{attribute 'GeneratedUsingTerminal: EL6201-0000-0017'}
{attribute addProperty BoxType "EL6201-0000-0017"}
{attribute addProperty Id "Slave_29A_DI0BOOL1Slave_29A_DI1BOOL1Slave_29A_DI2BOOL1Slave_29A_DI3BOOL1Slave_29B_DI0BOOL1Slave_29B_DI1BOOL1Slave_29B_DI2BOOL1Slave_29B_DI3BOOL1"}
{attribute addProperty CRC "3259051410"}
{attribute addProperty Size "8"}
TYPE Slave_29_Inputs_C2412D92 :
STRUCT
	{attribute addProperty Name "Slave_29A_DI0"}
	Slave_29A_DI0 : BOOL;
	{attribute addProperty Name "Slave_29A_DI1"}
	Slave_29A_DI1 : BOOL;
	{attribute addProperty Name "Slave_29A_DI2"}
	Slave_29A_DI2 : BOOL;
	{attribute addProperty Name "Slave_29A_DI3"}
	Slave_29A_DI3 : BOOL;
	{attribute addProperty Name "Slave_29B_DI0"}
	Slave_29B_DI0 : BOOL;
	{attribute addProperty Name "Slave_29B_DI1"}
	Slave_29B_DI1 : BOOL;
	{attribute addProperty Name "Slave_29B_DI2"}
	Slave_29B_DI2 : BOOL;
	{attribute addProperty Name "Slave_29B_DI3"}
	Slave_29B_DI3 : BOOL;
END_STRUCT
END_TYPE

(* stored: Version 1.2.0.0, ProductVersion 3.1.4024.9
   DUT Slave_29_Inputs_C2412D92: Id {317c4f93-2eeb-44ef-989c-eed3d043546f} *)
